# EPICS substitutions: beckhoffApp/Db/per_controller.substitutions
file "$(TOP)/beckhoffApp/beckhoff_read_pv.template" {
    pattern {P, NAME, PORT, ADSPORT, V, RECTYPE, EPICSDTYP, ADS_TYPE}
    {"\$(P)", "AXIS_NUM", "\$(PORT)", "\$(ADSPORT)", "GVL_APP.nAXIS_NUM", "longin", "asynInt32", "BOOL"}
}

file "$(TOP)/beckhoffApp/beckhoff_soft_pv.template" {
    pattern {P, NAME, VALUE, RECTYPE}
    {"\$(P)", "MTRCTRL", "\$(MTRCTRL)", "stringin"}
}
